// TIA Portal V19 export
TYPE "C402_STU_IF_SBO_TYPIC"
   STRUCT
      CMD_OPEN { ExternalAccessible := 'False'; ExternalVisible := 'False'; ExternalWritable := 'False'} : Bool;   // Aansturing afsluitboom Open
      CMD_VWA_TOE { ExternalAccessible := 'False'; ExternalVisible := 'False'; ExternalWritable := 'False'} : Bool;   // Aansturing afsluitboom voorwaardelijk Dicht
      CMD_TOE { ExternalAccessible := 'False'; ExternalVisible := 'False'; ExternalWritable := 'False'} : Bool;   // Aansturing afsluitboom (onvoorwaardelijk) Dicht
      CMD_STOP { ExternalAccessible := 'False'; ExternalVisible := 'False'; ExternalWritable := 'False'} : Bool;   // Aansturing afsluitboom Stop
      CMD_RES { ExternalAccessible := 'False'; ExternalVisible := 'False'; ExternalWritable := 'False'} : Bool;   // Reset van de latched storingen
      VGV_SNEL { ExternalAccessible := 'False'; ExternalVisible := 'False'; ExternalWritable := 'False'} : Bool;   // Vrijgave om versneld te sluiten
   END_STRUCT;
END_TYPE
